FUNCTION_BLOCK FB_AxisTemperature
VAR_INPUT
    bFbEnable: BOOL := FALSE;
    nAxisID: UINT;
    fMaxTemperature: LREAL := 0;
    nTempScalingFactor: INT := 10;
END_VAR
VAR_OUTPUT
    bFbEnabled: BOOL;
    fTemperatureValue: LREAL;
    bError: BOOL;
    sErrorMessage: STRING;
END_VAR
VAR
    eTemperatureStates: (eInit := 0, eError := 1, eRun := 2, eFbDisabled := 3):=0;
    nTempPT100 AT %I*: INT;
    sErrorMessageAxis: STRING;
    fbErrorTrig: R_TRIG;
    fbErrorTON: TON;
END_VAR

bFbEnabled := bFbEnable;
sErrorMessageAxis := CONCAT('ERROR: Temparture sensor of axis',INT_TO_STRING(nAxisID));

CASE eTemperatureStates OF
    eInit:
        IF NOT bFbEnabled THEN
            eTemperatureStates := eFbDisabled;
        ELSIF fTemperatureValue >= 85.0 OR fTemperatureValue <= -200.0 THEN
            eTemperatureStates := eError;
        ELSE
            eTemperatureStates := eRun;
        END_IF

    eError:

        GVL.astAxes[nAxisID].stStatus.fActTemperature := nTempPT100;
        GVL.astAxes[nAxisID].stStatus.bHighTempAxisDisabled := TRUE;
        fbErrorTrig(clk:=bError);
        fbErrorTON(in:=bError, PT:=T#10S);
        bError := TRUE;

        IF fbErrorTrig.Q THEN
            IF fTemperatureValue >= 85.0 THEN
                sErrorMessage := CONCAT(sErrorMessageAxis,' is disconnected');
                ADSLOGSTR( msgCtrlMask := ADSLOG_MSGTYPE_ERROR, msgFmtStr := '%s', strArg := sErrorMessage);
            ELSIF fTemperatureValue <= -200.0 THEN
                sErrorMessage := CONCAT(sErrorMessageAxis,' is wrongly connected, check PT100 pin connections');
                ADSLOGSTR( msgCtrlMask := ADSLOG_MSGTYPE_ERROR, msgFmtStr := '%s', strArg := sErrorMessage);
            END_IF
        END_IF

        //Reset bError to display Error message every 10 seconds if error is still there
        IF fbErrorTON.Q THEN
                bError := FALSE;
        END_IF

        eTemperatureStates := eInit;

    eRun:
        bError := FALSE;
        sErrorMessage := '';

        //Scale nTempPT100
        fTemperatureValue := nTempPT100 / nTempScalingFactor;
        IF fMaxTemperature = 0 OR fTemperatureValue < fMaxTemperature THEN
                GVL.astAxes[nAxisID].stStatus.bHighTempAxisDisabled := FALSE;
        ELSIF fTemperatureValue >= fMaxTemperature THEN
            GVL.astAxes[nAxisID].stStatus.bHighTempAxisDisabled := TRUE;
        END_IF

        eTemperatureStates := eInit;

    eFbDisabled:
        GVL.astAxes[nAxisID].stStatus.fActTemperature := 9999.0;
        GVL.astAxes[nAxisID].stStatus.bHighTempAxisDisabled := FALSE;
        bError := FALSE;
        sErrorMessage := '';

        IF NOT bFbEnabled THEN
            eTemperatureStates := eFbDisabled;
        ELSE
            eTemperatureStates := eInit;
        END_IF

END_CASE

END_FUNCTION_BLOCK

(* stored: Version 1.1.0.1, ProductVersion 3.1.4024.11
   POU FB_AxisTemperature: Id {dc25bdc5-b5d1-4653-9dd0-c72d7f39ce24}, SpecialFunc None *)
